{attribute 'GeneratedUsingTerminal: KL8001'}
{attribute addProperty BoxType "KL8001"}
{attribute addProperty Id "State_0AT %I*USINT0Data_In_0AT %I*UINT0State_1AT %I*USINT0Data_In_1AT %I*UINT0State_2AT %I*USINT0Data_In_2AT %I*UINT0State_ExtAT %I*USINT0Ctrl_0AT %Q*USINT0Data_Out_0AT %Q*UINT0Ctrl_1AT %Q*USINT0Data_Out_1AT %Q*UINT0Ctrl_2AT %Q*USINT0Data_Out_2AT %Q*UINT0Ctrl_ExtAT %Q*USINT0"}
{attribute addProperty CRC "3654584327"}
{attribute addProperty Size "0"}
TYPE Channel_D9D48807 :
STRUCT
	{attribute addProperty Name "State_0"}
	State_0 AT %I* : USINT;
	{attribute addProperty Name "Data_In_0"}
	Data_In_0 AT %I* : UINT;
	{attribute addProperty Name "State_1"}
	State_1 AT %I* : USINT;
	{attribute addProperty Name "Data_In_1"}
	Data_In_1 AT %I* : UINT;
	{attribute addProperty Name "State_2"}
	State_2 AT %I* : USINT;
	{attribute addProperty Name "Data_In_2"}
	Data_In_2 AT %I* : UINT;
	{attribute addProperty Name "State_Ext"}
	State_Ext AT %I* : USINT;
	{attribute addProperty Name "Ctrl_0"}
	Ctrl_0 AT %Q* : USINT;
	{attribute addProperty Name "Data_Out_0"}
	Data_Out_0 AT %Q* : UINT;
	{attribute addProperty Name "Ctrl_1"}
	Ctrl_1 AT %Q* : USINT;
	{attribute addProperty Name "Data_Out_1"}
	Data_Out_1 AT %Q* : UINT;
	{attribute addProperty Name "Ctrl_2"}
	Ctrl_2 AT %Q* : USINT;
	{attribute addProperty Name "Data_Out_2"}
	Data_Out_2 AT %Q* : UINT;
	{attribute addProperty Name "Ctrl_Ext"}
	Ctrl_Ext AT %Q* : USINT;
END_STRUCT
END_TYPE

(* stored: Version 1.2.0.0, ProductVersion 3.1.4024.9
   DUT Channel_D9D48807: Id {a0b8dbeb-4aa1-4432-9d10-44462766df84} *)
